(* Logix 5000 project; controller FTOptix_Datalog_trigger vendor 1 type 14 code 222 rev 36.11; software revision 36.00 *)

TASK MainTask (continuous, watchdog 500 ms) : MainProgram
TASK SafetyTask (periodic, rate 20 ms, priority 10, watchdog 20 ms, safety) : SafetyProgram

MODULES
   Local : vendor 1 type 14 code 222 (5069 0, rev 36.11)
END_MODULES

VAR_GLOBAL   (* controller tags *)
   PLC_Trigger : BOOL;
   Temperature : DINT;
   VariableToSample1 : DINT := 50;
   VariableToSample2 : DINT := 20;
   VariableToSample3 : DINT := 30;
   VariableToSample4 : DINT := 40;
   VariableToSample5 : DINT := 50;
   VariableToSample6 : DINT := 60;
END_VAR

PROGRAM MainProgram   (* main routine MainRoutine *)

ROUTINE MainRoutine   (* ladder *)
END_ROUTINE
END_PROGRAM

PROGRAM SafetyProgram   (* main routine MainRoutine, safety *)

ROUTINE MainRoutine   (* ladder *)
END_ROUTINE
END_PROGRAM
